(* Logix 5000 project; controller DUNEW2PLC1 vendor 1 type 14 code 221 rev 33.11; software revision 33.00; part 7 of 7 *)
(* tags used below, declared in another part *)
   current_command : REAL;
   current_command_high : REAL;
   current_command_low : REAL;
   ERROR_CODE : DINT;
   INIT_DONE : BOOL;
   max_tolerable_tension : REAL;
   MORE_STATS : BOOL[32];
   MOVE_TYPE : INT;   // 0 = No Move 1 = XY JOG 2 = XY Plane Move 3 = Z JOG 4 = Z Axis Move 5 = Toggle Latch Actuator 6 = Home the Latch Actuator
   neutral_cv : REAL;
   NEXTSTATE : DINT;
   overtension_timer : TIMER;
   pid_cv_high_limit : REAL;
   pid_cv_low_limit : REAL;
   PID_LOOP_TIMER : TIMER;
   Safety_Tripped_S : BOOL;
   STATE : DINT;   // CURRENT State Machine State
   STATE_REQUEST : DINT;
   tension : REAL;   // wire tension from load cell (N)
   TENSION_CONTROL_OK : BOOL;
   tension_motor_curr_override : REAL;
   tension_motor_cv : REAL;
   tension_off_oneshot : BOOL;
   tension_on_oneshot : BOOL;
   TENSION_ON_SWITCH : BOOL;
   tension_on_switch_delay_on_start : TIMER;
   tension_setpoint : REAL;
   tension_stable_timer : TIMER;
   tension_tag : ALIAS FOR Local:4:I.Ch01.Data;   // wire tension (N)
   winding_head_pid : PID;
   wire_broken_tension : REAL;
   wire_tensioned : BOOL;
   X_axis : AXIS_CIP_DRIVE;
   Y_axis : AXIS_CIP_DRIVE;
   Z_axis : AXIS_CIP_DRIVE;

PROGRAM state_9_unservo   (* main routine main *)
VAR
   entered_state_9_osr : BOOL;
   state_unservo_active : BOOL;
   unservo_ons_storage : BOOL[32];
   x_axis_mafr : MOTION_INSTRUCTION;
   x_axis_msf : MOTION_INSTRUCTION;
   x_axis_msf_dn_osr : BOOL;
   X_AXIS_STAT : MOTION_INSTRUCTION[32] := ([0].FLAGS := 570425344, [0].DN := 1, [0].STATUS := 2, [0].STATE := 1, [1].FLAGS := 570425344, [1].DN := 1, [1].STATE := 1, [2].FLAGS := 536870912, [2].DN := 1, [2].STATE := 1); {access Read Only}
   y_axis_mafr : MOTION_INSTRUCTION;
   y_axis_msf : MOTION_INSTRUCTION;
   y_axis_msf_dn_osr : BOOL;
   Y_AXIS_STAT : MOTION_INSTRUCTION[32] := ([0].FLAGS := 570425344, [0].DN := 1, [0].STATUS := 2, [0].STATE := 1, [1].FLAGS := 570425344, [1].DN := 1, [1].STATE := 1, [2].FLAGS := 536870912, [2].DN := 1, [2].STATE := 1); {access Read Only}
   z_axis_mafr : MOTION_INSTRUCTION;
   z_axis_msf : MOTION_INSTRUCTION;
   z_axis_msf_dn_osr : BOOL;
   Z_AXIS_STAT : MOTION_INSTRUCTION[32] := ([0].FLAGS := 570425344, [0].DN := 1, [0].STATUS := 2, [0].STATE := 1, [1].FLAGS := 570425344, [1].DN := 1, [1].STATE := 1, [2].FLAGS := 536870912, [2].DN := 1, [2].STATE := 1); {access Read Only}
END_VAR

ROUTINE main   (* ladder *)
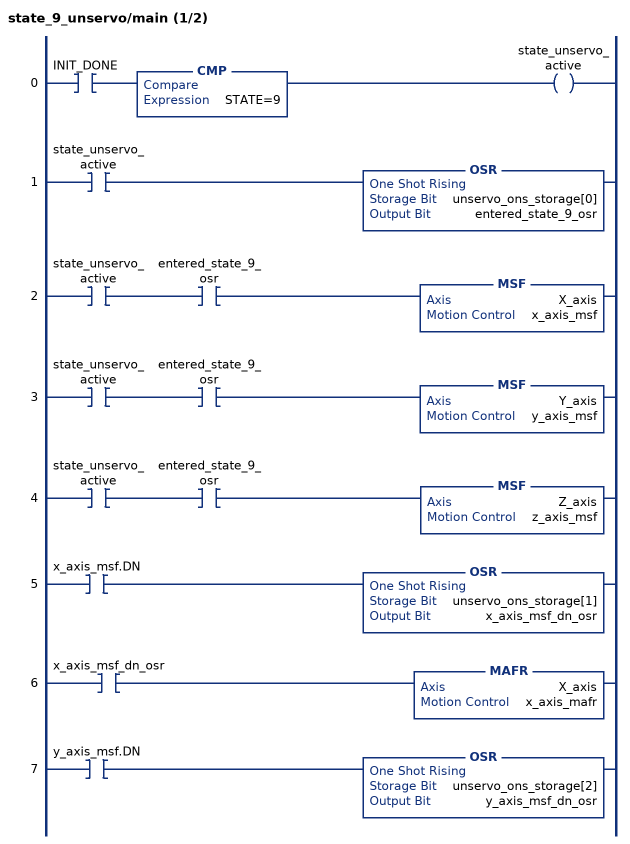
   0: XIC(INIT_DONE)CMP(STATE=9)OTE(state_unservo_active);
   1: XIC(state_unservo_active)OSR(unservo_ons_storage[0],entered_state_9_osr);
   2: XIC(state_unservo_active)XIC(entered_state_9_osr)MSF(X_axis,x_axis_msf);
   3: XIC(state_unservo_active)XIC(entered_state_9_osr)MSF(Y_axis,y_axis_msf);
   4: XIC(state_unservo_active)XIC(entered_state_9_osr)MSF(Z_axis,z_axis_msf);
   5: XIC(x_axis_msf.DN)OSR(unservo_ons_storage[1],x_axis_msf_dn_osr);
   6: XIC(x_axis_msf_dn_osr)MAFR(X_axis,x_axis_mafr);
   7: XIC(y_axis_msf.DN)OSR(unservo_ons_storage[2],y_axis_msf_dn_osr);
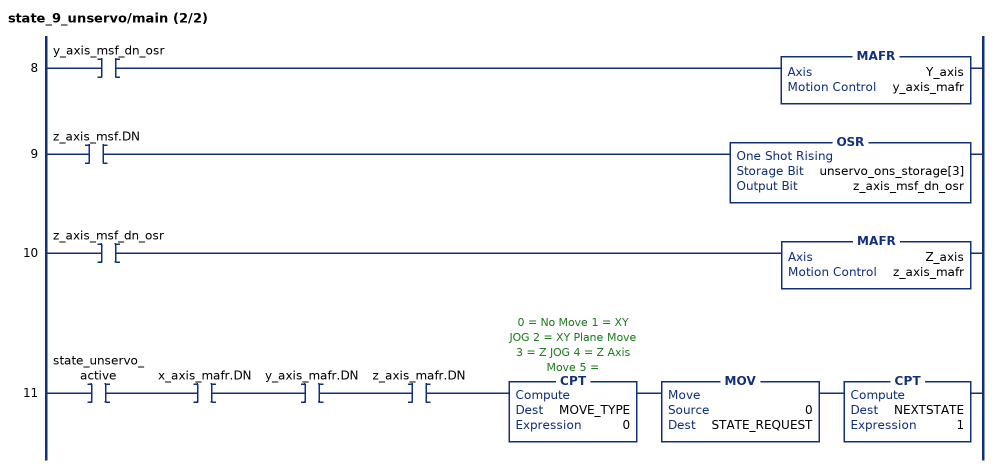
   8: XIC(y_axis_msf_dn_osr)MAFR(Y_axis,y_axis_mafr);
   9: XIC(z_axis_msf.DN)OSR(unservo_ons_storage[3],z_axis_msf_dn_osr);
   10: XIC(z_axis_msf_dn_osr)MAFR(Z_axis,z_axis_mafr);
   11: XIC(state_unservo_active)XIC(x_axis_mafr.DN)XIC(y_axis_mafr.DN)XIC(z_axis_mafr.DN)CPT(MOVE_TYPE,0)MOV(0,STATE_REQUEST)CPT(NEXTSTATE,1);
END_ROUTINE
END_PROGRAM

PROGRAM tension_pid   (* main routine main *)
// Using code from Sarah Johnson
VAR
   a0 : REAL := 0.6051849;
   a1 : REAL := 0.9277701;
   a2 : REAL;
   a3 : REAL;
   a4 : REAL;
   constant_cv_out : BOOL;
   cv_to_electrocraft : ALIAS FOR Local:5:O.Ch00.Data;
   disable_motor : BOOL := 1;
   Enable_tension_motor : ALIAS FOR Local:3:O.Pt03.Data;
   oneshotsb : BOOL[32] := ([0] := 1, [1] := 1);
   ramp_start_cv : REAL := 7.974453;
   tension_off_ramp_timer : TIMER := (PRE := 500);
   tension_stable_time : DINT := 10;
   tension_stable_tolerance : REAL := 0.2;
   wire_broke_osr_output_bit : BOOL;
   wire_broke_osr_storage_bit : BOOL;
   wire_broken_state : BOOL;
   wire_undertension_debounce : TIMER := (PRE := 1);
END_VAR

ROUTINE main   (* ladder *)
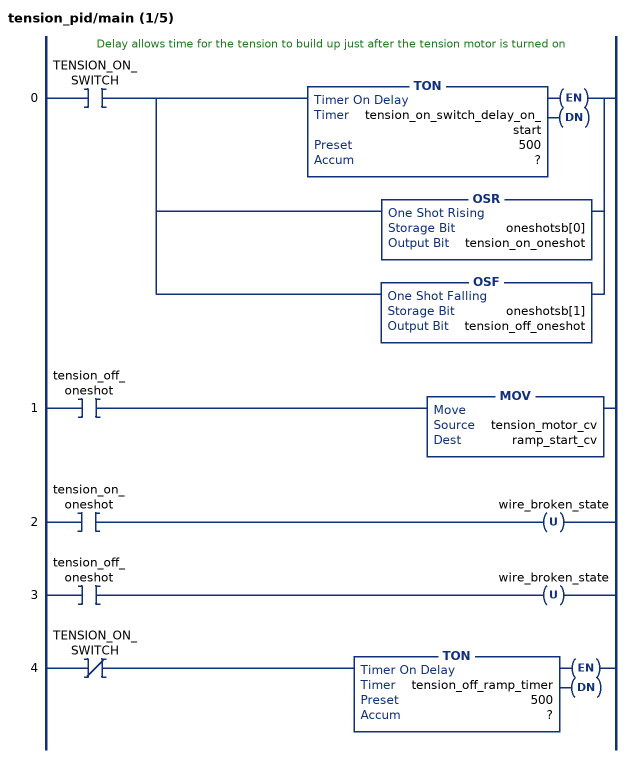
   // Delay allows time for the tension to build up just after the tension motor is turned on
   0: XIC(TENSION_ON_SWITCH)[TON(tension_on_switch_delay_on_start,?,?) ,OSR(oneshotsb[0],tension_on_oneshot) ,OSF(oneshotsb[1],tension_off_oneshot) ];
   1: XIC(tension_off_oneshot)MOV(tension_motor_cv,ramp_start_cv);
   2: XIC(tension_on_oneshot)OTU(wire_broken_state);
   3: XIC(tension_off_oneshot)OTU(wire_broken_state);
   4: XIO(TENSION_ON_SWITCH)TON(tension_off_ramp_timer,?,?);
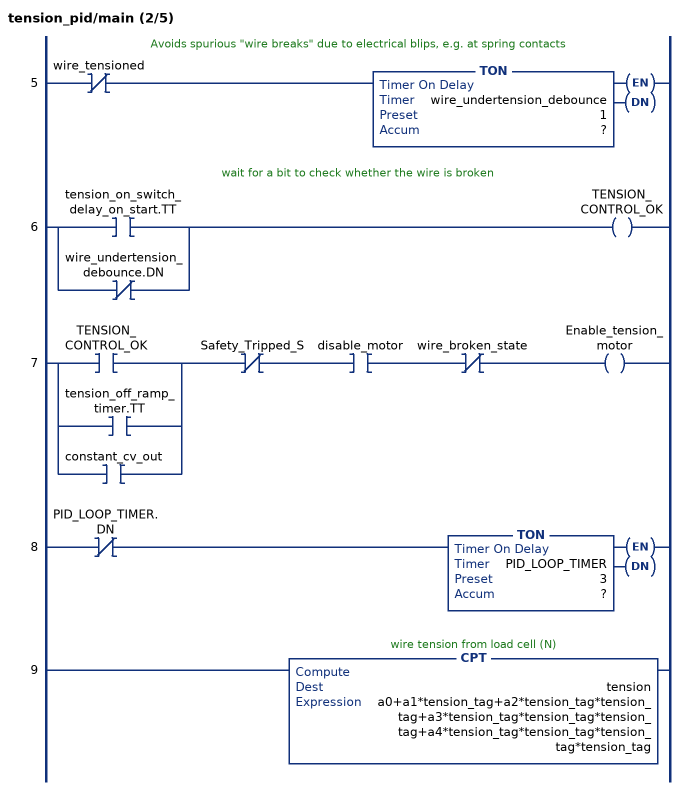
   // Avoids spurious "wire breaks" due to electrical blips, e.g. at spring contacts
   5: XIO(wire_tensioned)TON(wire_undertension_debounce,?,?);
   // wait for a bit to check whether the wire is broken
   6: [XIC(tension_on_switch_delay_on_start.TT) ,XIO(wire_undertension_debounce.DN) ]OTE(TENSION_CONTROL_OK);
   7: [XIC(TENSION_CONTROL_OK) ,XIC(tension_off_ramp_timer.TT) ,XIC(constant_cv_out) ]XIO(Safety_Tripped_S)XIC(disable_motor)XIO(wire_broken_state)OTE(Enable_tension_motor);
   8: XIO(PID_LOOP_TIMER.DN)TON(PID_LOOP_TIMER,?,?);
   9: CPT(tension,a0+a1*tension_tag+a2*tension_tag*tension_tag+a3*tension_tag*tension_tag*tension_tag+a4*tension_tag*tension_tag*tension_tag*tension_tag);
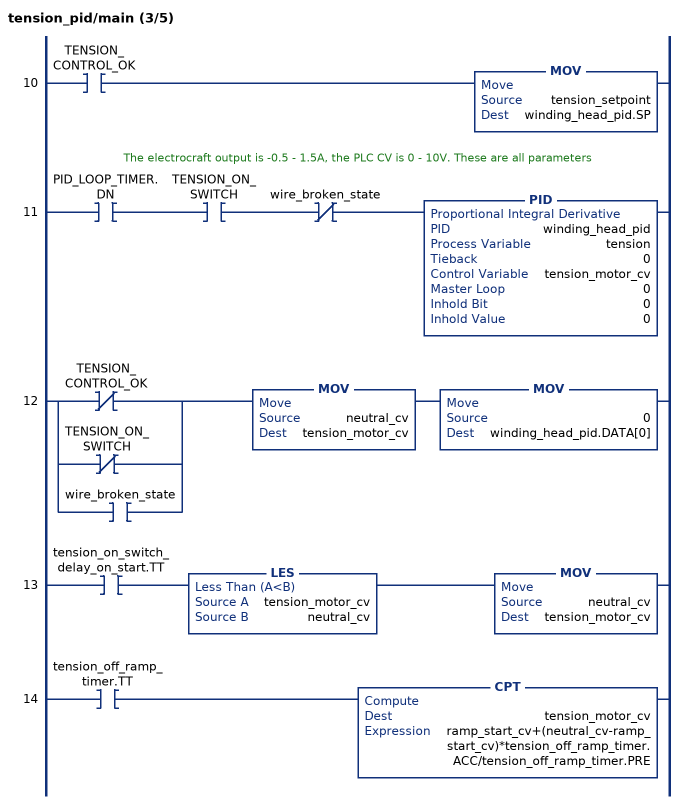
   10: XIC(TENSION_CONTROL_OK)MOV(tension_setpoint,winding_head_pid.SP);
   // The electrocraft output is -0.5 - 1.5A, the PLC CV is 0 - 10V. These are all parameters
   11: XIC(PID_LOOP_TIMER.DN)XIC(TENSION_ON_SWITCH)XIO(wire_broken_state)PID(winding_head_pid,tension,0,tension_motor_cv,0,0,0);
   12: [XIO(TENSION_CONTROL_OK) ,XIO(TENSION_ON_SWITCH) ,XIC(wire_broken_state) ]MOV(neutral_cv,tension_motor_cv)MOV(0,winding_head_pid.DATA[0]);
   13: XIC(tension_on_switch_delay_on_start.TT)LES(tension_motor_cv,neutral_cv)MOV(neutral_cv,tension_motor_cv);
   14: XIC(tension_off_ramp_timer.TT)CPT(tension_motor_cv,ramp_start_cv+(neutral_cv-ramp_start_cv)*tension_off_ramp_timer.ACC/tension_off_ramp_timer.PRE);
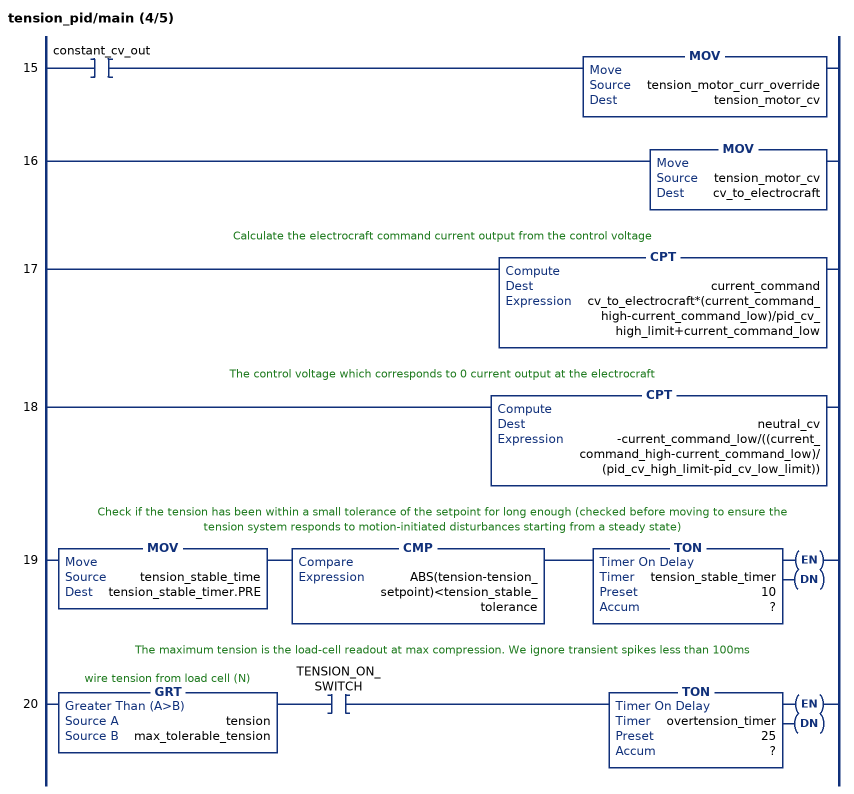
   15: XIC(constant_cv_out)MOV(tension_motor_curr_override,tension_motor_cv);
   16: MOV(tension_motor_cv,cv_to_electrocraft);
   // Calculate the electrocraft command current output from the control voltage
   17: CPT(current_command,cv_to_electrocraft*(current_command_high-current_command_low)/pid_cv_high_limit+current_command_low);
   // The control voltage which corresponds to 0 current output at the electrocraft
   18: CPT(neutral_cv,-current_command_low/((current_command_high-current_command_low)/(pid_cv_high_limit-pid_cv_low_limit)));
   // Check if the tension has been within a small tolerance of the setpoint for long enough (checked before moving to ensure the tension system responds to motion-initiated disturbances starting from a steady state)
   19: MOV(tension_stable_time,tension_stable_timer.PRE)CMP(ABS(tension-tension_setpoint)<tension_stable_tolerance)TON(tension_stable_timer,?,?);
   // The maximum tension is the load-cell readout at max compression. We ignore transient spikes less than 100ms
   20: GRT(tension,max_tolerable_tension)XIC(TENSION_ON_SWITCH)TON(overtension_timer,?,?);
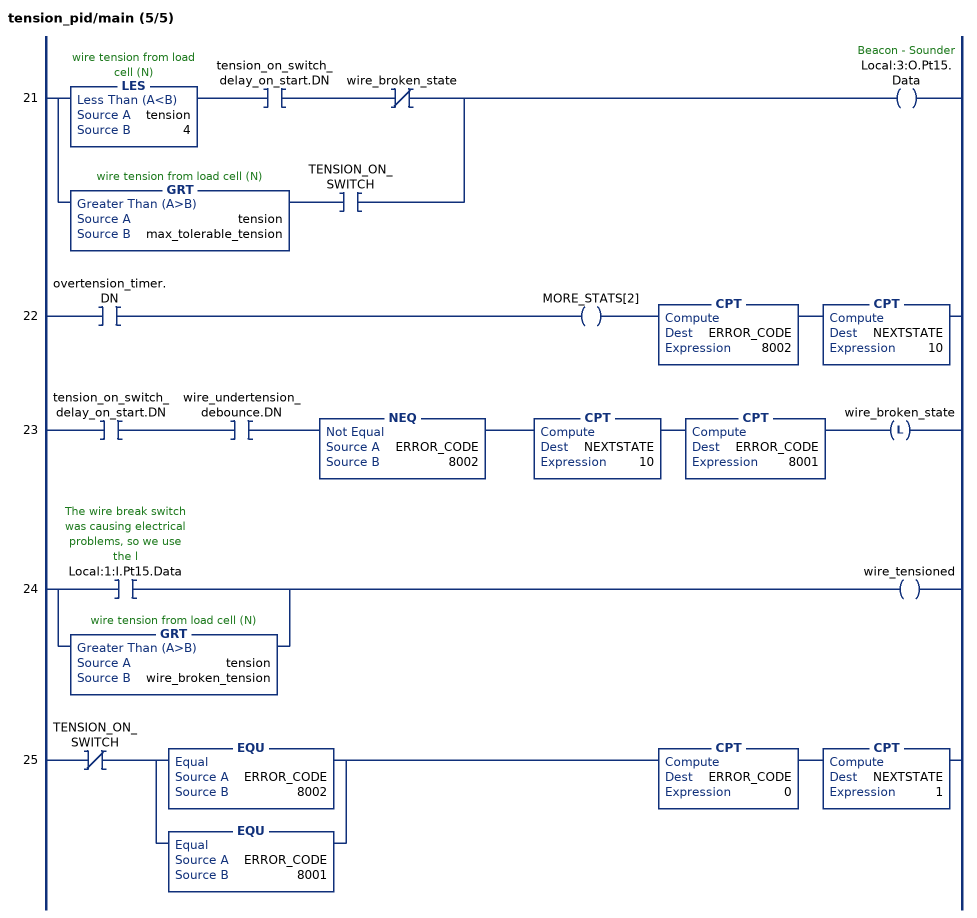
   21: [LES(tension,4) XIC(tension_on_switch_delay_on_start.DN) XIO(wire_broken_state) ,GRT(tension,max_tolerable_tension) XIC(TENSION_ON_SWITCH) ]OTE(Local:3:O.Pt15.Data);
   22: XIC(overtension_timer.DN)OTE(MORE_STATS[2])CPT(ERROR_CODE,8002)CPT(NEXTSTATE,10);
   23: XIC(tension_on_switch_delay_on_start.DN)XIC(wire_undertension_debounce.DN)NEQ(ERROR_CODE,8002)CPT(NEXTSTATE,10)CPT(ERROR_CODE,8001)OTL(wire_broken_state);
   24: [XIC(Local:1:I.Pt15.Data) ,GRT(tension,wire_broken_tension) ]OTE(wire_tensioned);
   25: XIO(TENSION_ON_SWITCH)[EQU(ERROR_CODE,8002) ,EQU(ERROR_CODE,8001) ]CPT(ERROR_CODE,0)CPT(NEXTSTATE,1);
END_ROUTINE
END_PROGRAM
